FUNCTION Buffer_Layout_Set_UInt_Array : UINT
VAR_INPUT
END_VAR
VAR
END_VAR

END_FUNCTION

(* stored: Version 1.1.0.1, ProductVersion 3.1.4024.10
   POU Buffer_Layout_Set_UInt_Array: Id {b7a1c8a9-e44c-4e03-8626-413f084fed49}, SpecialFunc None *)
